/// Implicitly generated code : DO NOT EDIT!!!
/// CheckBounds is used to check for range overflows
{attribute 'check_bounds' := ''}
{attribute 'no_check' := ''}
FUNCTION CheckBounds : DINT
VAR_INPUT
	index: DINT;
	lower: DINT;
	upper: DINT;
END_VAR

// align bounds 
CheckBounds := MIN(upper, MAX(lower, index));

// if index changed, report error
IF CheckBounds <> index THEN
	Services.fbEventHandler.Select(TC_Events.CodeEventClass.ErrorEvent)
						   .ArgSetString('check bounds')
						   .Raise();
END_IF

END_FUNCTION

(* stored: Version 1.1.0.1
   POU CheckBounds: Id {4909ba71-acf1-4751-90ca-8897514b75c2}, SpecialFunc None *)
